TYPE LrsPos :
STRUCT
	Pos:REAL;
	Height:REAL;
END_STRUCT
END_TYPE

(* stored: Version 1.1.0.1
   DUT LrsPos: Id {47bc8a4b-6b4a-4b98-b6e0-2b7c8867b492} *)
